KUKA KRL program: Rack_Azul_Inpicker.src, Rack_Azul_Inpicker.dat

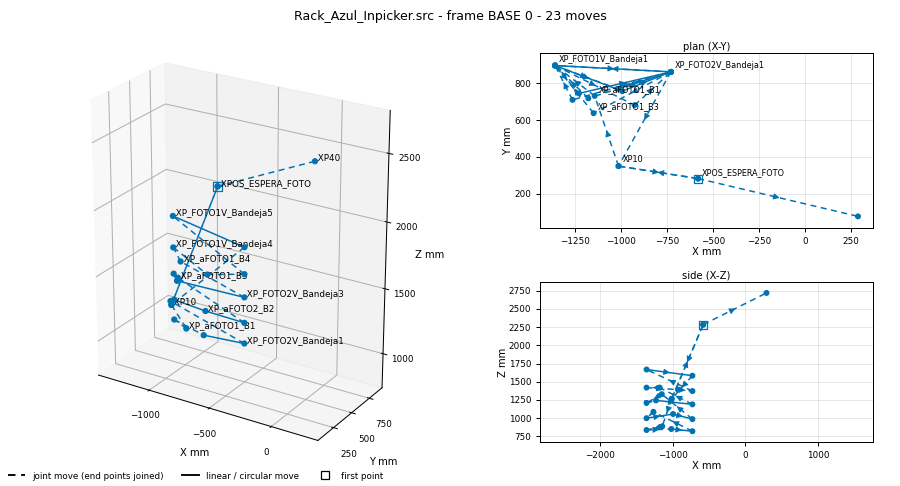
[picture p0: tool path of Rack_Azul_Inpicker.src in frame BASE 0, 23 of 23 moves have a stored position in this frame; points joined in program order, loops and branches not executed]
--- Rack_Azul_Inpicker.src ---
&ACCESS RVO1
&REL 136
&COMMENT FOTOS EN RACK AZUL
&PARAM EDITMASK = *
&PARAM TEMPLATE = C:\KRC\Roboter\Template\vorgabe
&PARAM DISKPATH = KRC:\R1\Program\MAFELEC
DEF Rack_Azul_Inpicker( )
;FOLD DECLARACION_INPICKER
DECL EKI_STATUS Ret
DECL INT InPickerStateValue
;ENDFOLD
;FOLD INI;%{PE}
  ;FOLD BASISTECH INI
    GLOBAL INTERRUPT DECL 3 WHEN $STOPMESS==TRUE DO IR_STOPM ( )
    INTERRUPT ON 3
    BAS (#INITMOV,0 )
  ;ENDFOLD (BASISTECH INI)
  ;FOLD USER INI
    ;Make your modifications here
O_LIMITS_OK=FALSE
O_LIMITS_NOK=FALSE
O_LIMIT_X=FALSE
O_LIMIT_Y=FALSE
O_LIMIT_Z=FALSE
O_LIMIT_A=FALSE
O_LIMIT_B=FALSE
O_LIMIT_C=FALSE
LIM_X=FALSE
LIM_Y=FALSE
LIM_Z=FALSE
LIM_A=FALSE
LIM_B=FALSE
LIM_C=FALSE
O_TYPE_INFO=0

  ;ENDFOLD (USER INI)
;ENDFOLD (INI)

;################################################
; PROYECTO: MAFELEC PLANTA DE BATERIAS
; ROBOT: 121_R1
; PROGRAMA: FOTO PARA CORRECCIONES EN RACK AZUL
; CREADO POR: Alejandro Company(zaisor robotics)
; FECHA: 23-NOVIEMBRE-2022
; MODIFICADO POR:
; FECHA MODIFICACION: 07-ENERO-2023
;################################################

;FOLD INICIALIZACION PUERTOS DE KRL
Ret = EKI_INIT("XML_Kuka_InPicker_1")
Ret = EKI_INIT("XML_Kuka_InPicker_2")

Ret = EKI_OPEN("XML_Kuka_InPicker_1")
Ret = EKI_OPEN("XML_Kuka_InPicker_2")

 INPICKER_Handler.DataToSend.command=0
;WAIT FOR (INPICKER_Handler.ConnectionStatus==TRUE)
;IF (INPICKER_Handler.ConnectionStatus==TRUE) THEN
;ELSE
;ENDIF

;ENDFOLD

Empujador(1,"R",FALSE)
Empujador(2,"R",FALSE)

; POSICION DE ESPERA ENTRADA RACK 2
;FOLD PTP POS_ESPERA_FOTO Vel=100 % H Tool[5]:T_Camara Base[0];%{PE}%R 8.3.48,%MKUKATPBASIS,%CMOVE,%VPTP,%P 1:PTP, 2:POS_ESPERA_FOTO, 3:, 5:100, 7:H
$BWDSTART=FALSE
PDAT_ACT=PH
FDAT_ACT=FPOS_ESPERA_FOTO
BAS(#PTP_PARAMS,100)
PTP XPOS_ESPERA_FOTO
;ENDFOLD

;ESPERA AREA 2
WAIT FOR I_ARDY_2
O_AREL_2=FALSE
RA_Bandeja_Nr=0

;FOLD PTP P10 CONT Vel=100 % M Tool[5]:T_Camara Base[0];%{PE}%R 8.3.48,%MKUKATPBASIS,%CMOVE,%VPTP,%P 1:PTP, 2:P10, 3:C_DIS, 5:100, 7:M
$BWDSTART=FALSE
PDAT_ACT=PM
FDAT_ACT=FP10
BAS(#PTP_PARAMS,100)
PTP XP10 C_DIS
;ENDFOLD
Empujador(1,"R",TRUE)
Empujador(2,"R",TRUE)

O_TYPE_RQ=TRUE
WAIT FOR (I_TYPE_INFO >= 20) AND (I_TYPE_INFO <= 26)

RA_Bandeja_Nr=I_TYPE_INFO

SWITCH RA_Bandeja_Nr

CASE 21
O_TYPE_INFO=RA_Bandeja_Nr
O_TYPE_RQ=FALSE
INICIO_FOTO1:
;FOLD PTP P_aFOTO1_B1 CONT Vel=50 % M Tool[5]:T_Camara Base[0];%{PE}%R 8.3.48,%MKUKATPBASIS,%CMOVE,%VPTP,%P 1:PTP, 2:P_aFOTO1_B1, 3:C_DIS, 5:50, 7:M
$BWDSTART=FALSE
PDAT_ACT=PM
FDAT_ACT=FP_aFOTO1_B1
BAS(#PTP_PARAMS,50)
PTP XP_aFOTO1_B1 C_DIS
;ENDFOLD
;FOLD PTP P_FOTO1V_Bandeja1 Vel=50 % M Tool[5]:T_Camara Base[0];%{PE}%R 8.3.48,%MKUKATPBASIS,%CMOVE,%VPTP,%P 1:PTP, 2:P_FOTO1V_Bandeja1, 3:, 5:50, 7:M
$BWDSTART=FALSE
PDAT_ACT=PM
FDAT_ACT=FP_FOTO1V_Bandeja1
BAS(#PTP_PARAMS,50)
PTP XP_FOTO1V_Bandeja1
;ENDFOLD
;FOLD REALIZA FOTO 1 BANDEJA 1
WAIT SEC 1.0
Fallo_nr=0
Ini1:
O_INPICKER_OK = FALSE
O_INPICKER_NOK = FALSE
SELECT_SIN=FALSE
SELECT_U1=FALSE
SELECT_U2=FALSE
SELECT_U3=FALSE
SELECT_U4=FALSE

; INICIALIZACION CAMARA PARA BANDEJA 1
 INPICKER_Handler.DataToSend.command=0
 INPICKER_Handler.DataToSend.GraspConfirmation=0
 WAIT FOR (INPICKER_Handler.DataReceived.state==0)

; Camara siempre 2
 INPICKER_Handler.DataToSend.CameraID=2

; contendor igual al numero de bandeja
 INPICKER_Handler.DataToSend.ContainerID=6
 INPICKER_Handler.DataToSend.partid=6
 INPICKER_Handler.DataToSend.GraspConfirmation=0
 WAIT SEC 0.2

; DISPARO FOTO
 INPICKER_Handler.DataToSend.command=1

; ESPERA FOTO REALIZADA
 WAIT FOR (INPICKER_Handler.DataReceived.state==15) OR (INPICKER_Handler.DataReceived.state==-1)

IF (INPICKER_Handler.DataReceived.state==-1) THEN

IF (Fallo_nr>=1) THEN
O_INPICKER_OK=FALSE
O_INPICKER_NOK=TRUE

O_TYPE_RQ = FALSE
WAIT FOR I_TYPE_INFO == 0

O_TYPE_RQ = TRUE
WAIT FOR (I_TYPE_INFO >= 1) AND (I_TYPE_INFO <= 5)

SWITCH I_TYPE_INFO

CASE 2
; #### SELECCION DESDE HMI REINTENTO FOTO ####

SELECT_NEXT=FALSE
O_INPICKER_OK=FALSE
O_INPICKER_NOK=FALSE
O_TYPE_RQ = FALSE
GOTO Ini1

CASE 3
; #### SELECCION DESDE HMI CONT SIN CORRECCION ####

SELECT_SIN=TRUE
O_INPICKER_OK=FALSE
O_INPICKER_NOK=TRUE
O_TYPE_RQ = FALSE
GOTO FIN_FOTO1

CASE 4
; #### SELECCION DESDE HMI CERRAR BANDEJA ####
; #### E IR A SIGUIENTE NIVEL             ####

SELECT_NEXT=TRUE
O_INPICKER_OK=FALSE
O_INPICKER_NOK=FALSE
O_TYPE_RQ = FALSE
GOTO FIN_FOTO1

DEFAULT
ENDSWITCH

ELSE

Fallo_nr=Fallo_nr+1
GOTO Ini1

ENDIF
ENDIF

Fin1:
 WAIT SEC 0.1
;ENDFOLD

;FOLD PTP P_aFOTO2_B1 CONT Vel=50 % M Tool[5]:T_Camara Base[0];%{PE}%R 8.3.48,%MKUKATPBASIS,%CMOVE,%VPTP,%P 1:PTP, 2:P_aFOTO2_B1, 3:C_DIS, 5:50, 7:M
$BWDSTART=FALSE
PDAT_ACT=PM
FDAT_ACT=FP_aFOTO2_B1
BAS(#PTP_PARAMS,50)
PTP XP_aFOTO2_B1 C_DIS
;ENDFOLD

;FOLD LIN P_FOTO2V_Bandeja1 Vel=0.5 m/s M Tool[5]:T_Camara Base[0];%{PE}%R 8.3.48,%MKUKATPBASIS,%CMOVE,%VLIN,%P 1:LIN, 2:P_FOTO2V_Bandeja1, 3:, 5:0.5, 7:M
$BWDSTART=FALSE
LDAT_ACT=LM
FDAT_ACT=FP_FOTO2V_Bandeja1
BAS(#CP_PARAMS,0.5)
LIN XP_FOTO2V_Bandeja1
;ENDFOLD
;FOLD REALIZA FOTO 2 BANDEJA 1 (INFERIOR)
WAIT SEC 1.0
INPICKER_Handler.DataToSend.GraspConfirmation=1

WAIT FOR (INPICKER_Handler.DataReceived.state==30) OR (INPICKER_Handler.dataReceived.state==-1)
WAIT SEC 0.5

INPICKER_Handler.DataToSend.command=0

IF (INPICKER_handler.datareceived.state==30 ) THEN

IF (INPICKER_Handler.DataReceived.ObjectsGraspable>0) THEN

O_INPICKER_OK=TRUE
O_INPICKER_NOK=FALSE

ELSE

O_INPICKER_OK=FALSE
O_INPICKER_NOK=TRUE

ENDIF

ENDIF

IF (INPICKER_handler.datareceived.state==-1 ) OR (INPICKER_Handler.DataReceived.ObjectsGraspable<=0) THEN

O_INPICKER_OK=FALSE
O_INPICKER_NOK=TRUE

O_TYPE_RQ = FALSE
WAIT FOR I_TYPE_INFO == 0

O_TYPE_RQ = TRUE
WAIT FOR (I_TYPE_INFO >= 1) AND (I_TYPE_INFO <= 5)

SWITCH I_TYPE_INFO

CASE 2
; #### SELECCION DESDE HMI REINTENTO FOTO ####

SELECT_NEXT=FALSE
O_INPICKER_OK=FALSE
O_INPICKER_NOK=FALSE
O_TYPE_RQ = FALSE

IF (INPICKER_Handler.DataReceived.ObjectsGraspable>0)THEN
ELSE
GOTO INICIO_FOTO1
ENDIF

WAIT FOR (INPICKER_Handler.DataReceived.state==0)
GOTO INICIO_FOTO1

CASE 3
; #### SELECCION DESDE HMI CONT SIN CORRECCION ####

SELECT_NEXT=FALSE
O_TYPE_RQ = FALSE

CASE 4
; #### SELECCION DESDE HMI CERRAR BANDEJA ####
; #### E IR A SIGUIENTE NIVEL             ####

SELECT_NEXT=TRUE
O_INPICKER_OK=FALSE
O_INPICKER_NOK=FALSE
O_TYPE_RQ = FALSE

DEFAULT
ENDSWITCH

ENDIF

;ENDFOLD
;FOLD ACTUALIZA BASE DE DESCARGA
FRAMEAUX={X 0,Y 0,Z 0,A 0,B 0,C 0}
FRAME_POS={X 0,Y 0,Z 0,A 0,B 0,C 0}

FRAMEAUX=INPICKER_Handler.DataReceived.PartsToGrasp0.Position
FRAME_POS.x=(FRAMEAUX.x/10)
FRAME_POS.y=(FRAMEAUX.y/10)
FRAME_POS.z=(FRAMEAUX.z/10)
FRAME_POS.a=(FRAMEAUX.a/10)
FRAME_POS.b=(FRAMEAUX.b/10)
FRAME_POS.c=(FRAMEAUX.c/10)

IF FRAME_POS.A < 180.0 THEN
FRAME_POS.A = FRAME_POS.A + 360
ENDIF
IF FRAME_POS.B < 180.0 THEN
FRAME_POS.B = FRAME_POS.B + 360
ENDIF
IF FRAME_POS.A > 180.0 THEN
FRAME_POS.A = FRAME_POS.A - 360
ENDIF
IF FRAME_POS.B > 180.0 THEN
FRAME_POS.B = FRAME_POS.B - 360
ENDIF

FRAME_POS.C = FRAME_POS.C - 360

;ENDFOLD
;FOLD CONTROL LIMITES DE VISION
CTRL_limites()
;ENDFOLD
;FOLD DECISION RESULTADOS EVALUACION BANDEJA 1

IF (O_INPICKER_OK==FALSE) AND (O_INPICKER_NOK==TRUE) THEN
SELECT_NEXT=FALSE
O_TYPE_RQ = FALSE
GOTO FIN_FOTO1
ENDIF


IF (O_LIMITS_OK==FALSE) AND (O_LIMITS_NOK==TRUE) THEN

O_TYPE_RQ = FALSE
WAIT FOR I_TYPE_INFO == 0

O_TYPE_RQ = TRUE
WAIT FOR (I_TYPE_INFO >= 1) AND (I_TYPE_INFO <= 5)

SWITCH I_TYPE_INFO

CASE 2
; #### SELECCION DESDE HMI REINTENTO FOTO ####

SELECT_NEXT=FALSE
O_TYPE_RQ = FALSE
O_LIMITS_OK = FALSE
O_LIMITS_NOK = FALSE
O_LIMIT_X = FALSE
O_LIMIT_Y = FALSE
O_LIMIT_Z = FALSE
O_LIMIT_A = FALSE
O_LIMIT_B = FALSE
O_LIMIT_C = FALSE

GOTO INICIO_FOTO1

CASE 3
; #### SELECCION DESDE HMI CONT SIN CORRECCION ####

SELECT_NEXT=FALSE
O_TYPE_RQ = FALSE

CASE 4
; #### SELECCION DESDE HMI CERRAR BANDEJA ####
; #### E IR A SIGUIENTE NIVEL             ####

SELECT_NEXT=TRUE
O_TYPE_RQ = FALSE
O_LIMITS_OK = FALSE
O_LIMITS_NOK = FALSE
O_LIMIT_X = FALSE
O_LIMIT_Y = FALSE
O_LIMIT_Z = FALSE
O_LIMIT_A = FALSE
O_LIMIT_B = FALSE
O_LIMIT_C = FALSE

DEFAULT

HALT
HALT
HALT
ENDSWITCH

ENDIF

NO_TYPE_LBL:
;ENDFOLD
FIN_FOTO1:

CASE 22
O_TYPE_INFO=RA_Bandeja_Nr
O_TYPE_RQ=FALSE
INICIO_FOTO2:
;FOLD PTP P_aFOTO1_B2 Vel=50 % M Tool[5]:T_Camara Base[0];%{PE}%R 8.3.48,%MKUKATPBASIS,%CMOVE,%VPTP,%P 1:PTP, 2:P_aFOTO1_B2, 3:, 5:50, 7:M
$BWDSTART=FALSE
PDAT_ACT=PM
FDAT_ACT=FP_aFOTO1_B2
BAS(#PTP_PARAMS,50)
PTP XP_aFOTO1_B2
;ENDFOLD
;FOLD PTP P_FOTO1V_Bandeja2 Vel=50 % M Tool[5]:T_Camara Base[0];%{PE}%R 8.3.48,%MKUKATPBASIS,%CMOVE,%VPTP,%P 1:PTP, 2:P_FOTO1V_Bandeja2, 3:, 5:50, 7:M
$BWDSTART=FALSE
PDAT_ACT=PM
FDAT_ACT=FP_FOTO1V_Bandeja2
BAS(#PTP_PARAMS,50)
PTP XP_FOTO1V_Bandeja2
;ENDFOLD
;FOLD REALIZA FOTO 1 BANDEJA 2
WAIT SEC 1.0
Fallo_nr=0
Ini2:
O_INPICKER_OK = FALSE
O_INPICKER_NOK = FALSE
SELECT_SIN=FALSE
SELECT_U1=FALSE
SELECT_U2=FALSE
SELECT_U3=FALSE
SELECT_U4=FALSE

; INICIALIZACION CAMARA PARA BANDEJA 2
 INPICKER_Handler.DataToSend.command=0
 INPICKER_Handler.DataToSend.GraspConfirmation=0
 WAIT FOR (INPICKER_Handler.DataReceived.state==0)

; Camara siempre 2
 INPICKER_Handler.DataToSend.CameraID=2

; contendor igual al numero de bandeja
 INPICKER_Handler.DataToSend.ContainerID=7
 INPICKER_Handler.DataToSend.partid=7
 INPICKER_Handler.DataToSend.GraspConfirmation=0
 WAIT SEC 0.2

; DISPARO FOTO
 INPICKER_Handler.DataToSend.command=1

; ESPERA FOTO REALIZADA
 WAIT FOR (INPICKER_Handler.DataReceived.state==15) OR (INPICKER_Handler.DataReceived.state==-1)

IF (INPICKER_Handler.DataReceived.state==-1) THEN

IF (Fallo_nr>=1) THEN
O_INPICKER_OK=FALSE
O_INPICKER_NOK=TRUE

O_TYPE_RQ = FALSE
WAIT FOR I_TYPE_INFO == 0

O_TYPE_RQ = TRUE
WAIT FOR (I_TYPE_INFO >= 1) AND (I_TYPE_INFO <= 5)

SWITCH I_TYPE_INFO

CASE 2
; #### SELECCION DESDE HMI REINTENTO FOTO ####

SELECT_NEXT=FALSE
O_INPICKER_OK=FALSE
O_INPICKER_NOK=FALSE
O_TYPE_RQ = FALSE
GOTO Ini2

CASE 3
; #### SELECCION DESDE HMI CONT SIN CORRECCION ####

SELECT_SIN=TRUE
O_INPICKER_OK=FALSE
O_INPICKER_NOK=TRUE
O_TYPE_RQ = FALSE
GOTO FIN_FOTO2

CASE 4
; #### SELECCION DESDE HMI CERRAR BANDEJA ####
; #### E IR A SIGUIENTE NIVEL             ####

SELECT_NEXT=TRUE
O_INPICKER_OK=FALSE
O_INPICKER_NOK=FALSE
O_TYPE_RQ = FALSE
GOTO FIN_FOTO2

DEFAULT
ENDSWITCH

ELSE

Fallo_nr=Fallo_nr+1
GOTO Ini2

ENDIF
ENDIF

Fin2:
 WAIT SEC 0.1
;ENDFOLD

;FOLD LIN P_aFOTO2_B2 Vel=0.3 m/s M Tool[5]:T_Camara Base[0];%{PE}%R 8.3.48,%MKUKATPBASIS,%CMOVE,%VLIN,%P 1:LIN, 2:P_aFOTO2_B2, 3:, 5:0.3, 7:M
$BWDSTART=FALSE
LDAT_ACT=LM
FDAT_ACT=FP_aFOTO2_B2
BAS(#CP_PARAMS,0.3)
LIN XP_aFOTO2_B2
;ENDFOLD

;FOLD LIN P_FOTO2V_Bandeja2 Vel=0.5 m/s M Tool[5]:T_Camara Base[0];%{PE}%R 8.3.48,%MKUKATPBASIS,%CMOVE,%VLIN,%P 1:LIN, 2:P_FOTO2V_Bandeja2, 3:, 5:0.5, 7:M
$BWDSTART=FALSE
LDAT_ACT=LM
FDAT_ACT=FP_FOTO2V_Bandeja2
BAS(#CP_PARAMS,0.5)
LIN XP_FOTO2V_Bandeja2
;ENDFOLD
;FOLD REALIZA FOTO 2 BANDEJA 2
WAIT SEC 1.0
INPICKER_Handler.DataToSend.GraspConfirmation=1

WAIT FOR (INPICKER_Handler.DataReceived.state==30) OR (INPICKER_Handler.dataReceived.state==-1)

WAIT SEC 0.5

INPICKER_Handler.DataToSend.command=0

IF (INPICKER_handler.datareceived.state==30 ) THEN

IF (INPICKER_Handler.DataReceived.ObjectsGraspable>0) THEN

O_INPICKER_OK=TRUE
O_INPICKER_NOK=FALSE

ELSE

O_INPICKER_OK=FALSE
O_INPICKER_NOK=TRUE

ENDIF

ENDIF

IF (INPICKER_handler.datareceived.state==-1 ) OR (INPICKER_Handler.DataReceived.ObjectsGraspable<=0) THEN

O_INPICKER_OK=FALSE
O_INPICKER_NOK=TRUE

O_TYPE_RQ = FALSE
WAIT FOR I_TYPE_INFO == 0

O_TYPE_RQ = TRUE
WAIT FOR (I_TYPE_INFO >= 1) AND (I_TYPE_INFO <= 5)

SWITCH I_TYPE_INFO

CASE 2
; #### SELECCION DESDE HMI REINTENTO FOTO ####

SELECT_NEXT=FALSE
O_INPICKER_OK=FALSE
O_INPICKER_NOK=FALSE
O_TYPE_RQ = FALSE

IF (INPICKER_Handler.DataReceived.ObjectsGraspable>0)THEN
ELSE
GOTO INICIO_FOTO2
ENDIF

WAIT FOR (INPICKER_Handler.DataReceived.state==0)
GOTO INICIO_FOTO2

CASE 3
; #### SELECCION DESDE HMI CONT SIN CORRECCION ####

SELECT_NEXT=FALSE
O_TYPE_RQ = FALSE

CASE 4
; #### SELECCION DESDE HMI CERRAR BANDEJA ####
; #### E IR A SIGUIENTE NIVEL             ####

SELECT_NEXT=TRUE
O_INPICKER_OK=FALSE
O_INPICKER_NOK=FALSE
O_TYPE_RQ = FALSE

DEFAULT
ENDSWITCH

ENDIF

;ENDFOLD
;FOLD ACTUALIZA BASE DE DESCARGA
FRAMEAUX={X 0,Y 0,Z 0,A 0,B 0,C 0}
FRAME_POS={X 0,Y 0,Z 0,A 0,B 0,C 0}

FRAMEAUX=INPICKER_Handler.DataReceived.PartsToGrasp0.Position
FRAME_POS.x=(FRAMEAUX.x/10)
FRAME_POS.y=(FRAMEAUX.y/10)
FRAME_POS.z=(FRAMEAUX.z/10)
FRAME_POS.a=(FRAMEAUX.a/10)
FRAME_POS.b=(FRAMEAUX.b/10)
FRAME_POS.c=(FRAMEAUX.c/10)

IF FRAME_POS.A < 180.0 THEN
FRAME_POS.A = FRAME_POS.A + 360
ENDIF
IF FRAME_POS.B < 180.0 THEN
FRAME_POS.B = FRAME_POS.B + 360
ENDIF
IF FRAME_POS.A > 180.0 THEN
FRAME_POS.A = FRAME_POS.A - 360
ENDIF
IF FRAME_POS.B > 180.0 THEN
FRAME_POS.B = FRAME_POS.B - 360
ENDIF
FRAME_POS.C = FRAME_POS.C - 360
;ENDFOLD
;FOLD CONTROL LIMITES DE VISION
CTRL_limites()
;ENDFOLD
;FOLD DECISION RESULTADOS EVALUACION BANDEJA 2

IF (O_INPICKER_OK==FALSE) AND (O_INPICKER_NOK==TRUE) THEN
SELECT_NEXT=FALSE
O_TYPE_RQ = FALSE
GOTO FIN_FOTO2
ENDIF



IF (O_LIMITS_OK==FALSE) AND (O_LIMITS_NOK==TRUE) THEN

O_TYPE_RQ = FALSE
WAIT FOR I_TYPE_INFO == 0

O_TYPE_RQ = TRUE
WAIT FOR (I_TYPE_INFO >= 1) AND (I_TYPE_INFO <= 5)

SWITCH I_TYPE_INFO

CASE 2
; #### SELECCION DESDE HMI REINTENTO FOTO ####

SELECT_NEXT=FALSE
O_TYPE_RQ = FALSE
O_LIMITS_OK = FALSE
O_LIMITS_NOK = FALSE
O_LIMIT_X = FALSE
O_LIMIT_Y = FALSE
O_LIMIT_Z = FALSE
O_LIMIT_A = FALSE
O_LIMIT_B = FALSE
O_LIMIT_C = FALSE

GOTO INICIO_FOTO2

CASE 3
; #### SELECCION DESDE HMI CONT SIN CORRECCION ####

SELECT_NEXT=FALSE
O_TYPE_RQ = FALSE

CASE 4
; #### SELECCION DESDE HMI CERRAR BANDEJA ####
; #### E IR A SIGUIENTE NIVEL             ####

SELECT_NEXT=TRUE
O_TYPE_RQ = FALSE
O_LIMITS_OK = FALSE
O_LIMITS_NOK = FALSE
O_LIMIT_X = FALSE
O_LIMIT_Y = FALSE
O_LIMIT_Z = FALSE
O_LIMIT_A = FALSE
O_LIMIT_B = FALSE
O_LIMIT_C = FALSE

DEFAULT

HALT
HALT
HALT
ENDSWITCH

ENDIF

;ENDFOLD
FIN_FOTO2:

CASE 23
O_TYPE_RQ=FALSE
O_TYPE_INFO=RA_Bandeja_Nr
INICIO_FOTO3:
;FOLD PTP P_aFOTO1_B3 CONT Vel=50 % M Tool[5]:T_Camara Base[0];%{PE}%R 8.3.48,%MKUKATPBASIS,%CMOVE,%VPTP,%P 1:PTP, 2:P_aFOTO1_B3, 3:C_DIS, 5:50, 7:M
$BWDSTART=FALSE
PDAT_ACT=PM
FDAT_ACT=FP_aFOTO1_B3
BAS(#PTP_PARAMS,50)
PTP XP_aFOTO1_B3 C_DIS
;ENDFOLD
;FOLD PTP P_FOTO1V_Bandeja3 Vel=50 % M Tool[5]:T_Camara Base[0];%{PE}%R 8.3.48,%MKUKATPBASIS,%CMOVE,%VPTP,%P 1:PTP, 2:P_FOTO1V_Bandeja3, 3:, 5:50, 7:M
$BWDSTART=FALSE
PDAT_ACT=PM
FDAT_ACT=FP_FOTO1V_Bandeja3
BAS(#PTP_PARAMS,50)
PTP XP_FOTO1V_Bandeja3
;ENDFOLD
;FOLD REALIZA FOTO 1 BANDEJA 3
WAIT SEC 1.0
Fallo_nr=0
Ini3:
O_INPICKER_OK = FALSE
O_INPICKER_NOK = FALSE
SELECT_SIN=FALSE
SELECT_U1=FALSE
SELECT_U2=FALSE
SELECT_U3=FALSE
SELECT_U4=FALSE

; INICIALIZACION CAMARA PARA BANDEJA 3
 INPICKER_Handler.DataToSend.command=0
 INPICKER_Handler.DataToSend.GraspConfirmation=0
 WAIT FOR (INPICKER_Handler.DataReceived.state==0)

; Camara siempre 2
 INPICKER_Handler.DataToSend.CameraID=2

; contendor igual al numero de bandeja
 INPICKER_Handler.DataToSend.ContainerID=8
 INPICKER_Handler.DataToSend.partid=8
 INPICKER_Handler.DataToSend.GraspConfirmation=0
 WAIT SEC 0.2

; DISPARO FOTO
 INPICKER_Handler.DataToSend.command=1

; ESPERA FOTO REALIZADA
 WAIT FOR (INPICKER_Handler.DataReceived.state==15) OR (INPICKER_Handler.DataReceived.state==-1)

IF (INPICKER_Handler.DataReceived.state==-1) THEN

IF (Fallo_nr>=1) THEN
O_INPICKER_OK=FALSE
O_INPICKER_NOK=TRUE

O_TYPE_RQ = FALSE
WAIT FOR I_TYPE_INFO == 0

O_TYPE_RQ = TRUE
WAIT FOR (I_TYPE_INFO >= 1) AND (I_TYPE_INFO <= 5)

SWITCH I_TYPE_INFO

CASE 2
; #### SELECCION DESDE HMI REINTENTO FOTO ####

SELECT_NEXT=FALSE
O_INPICKER_OK=FALSE
O_INPICKER_NOK=FALSE
O_TYPE_RQ = FALSE
GOTO Ini3

CASE 3
; #### SELECCION DESDE HMI CONT SIN CORRECCION ####

SELECT_SIN=TRUE
O_INPICKER_OK=FALSE
O_INPICKER_NOK=TRUE
O_TYPE_RQ = FALSE
GOTO FIN_FOTO3

CASE 4
; #### SELECCION DESDE HMI CERRAR BANDEJA ####
; #### E IR A SIGUIENTE NIVEL             ####

SELECT_NEXT=TRUE
O_INPICKER_OK=FALSE
O_INPICKER_NOK=FALSE
O_TYPE_RQ = FALSE
GOTO FIN_FOTO3

DEFAULT
ENDSWITCH

ELSE

Fallo_nr=Fallo_nr+1
GOTO Ini3

ENDIF
ENDIF

Fin3:
 WAIT SEC 0.1
;ENDFOLD

;FOLD PTP P_aFOTO2_B3 CONT Vel=50 % M Tool[5]:T_Camara Base[0];%{PE}%R 8.3.48,%MKUKATPBASIS,%CMOVE,%VPTP,%P 1:PTP, 2:P_aFOTO2_B3, 3:C_DIS, 5:50, 7:M
$BWDSTART=FALSE
PDAT_ACT=PM
FDAT_ACT=FP_aFOTO2_B3
BAS(#PTP_PARAMS,50)
PTP XP_aFOTO2_B3 C_DIS
;ENDFOLD

;FOLD LIN P_FOTO2V_Bandeja3 Vel=0.3 m/s M Tool[5]:T_Camara Base[0];%{PE}%R 8.3.48,%MKUKATPBASIS,%CMOVE,%VLIN,%P 1:LIN, 2:P_FOTO2V_Bandeja3, 3:, 5:0.3, 7:M
$BWDSTART=FALSE
LDAT_ACT=LM
FDAT_ACT=FP_FOTO2V_Bandeja3
BAS(#CP_PARAMS,0.3)
LIN XP_FOTO2V_Bandeja3
;ENDFOLD
;FOLD REALIZA FOTO 2 BANDEJA 3
WAIT SEC 1.0
INPICKER_Handler.DataToSend.GraspConfirmation=1

WAIT FOR (INPICKER_Handler.DataReceived.state==30) OR (INPICKER_Handler.dataReceived.state==-1)

WAIT SEC 0.5

INPICKER_Handler.DataToSend.command=0

IF (INPICKER_handler.datareceived.state==30 ) THEN

IF (INPICKER_Handler.DataReceived.ObjectsGraspable>0) THEN

O_INPICKER_OK=TRUE
O_INPICKER_NOK=FALSE

ELSE

O_INPICKER_OK=FALSE
O_INPICKER_NOK=TRUE

ENDIF

ENDIF

IF (INPICKER_handler.datareceived.state==-1 ) OR (INPICKER_Handler.DataReceived.ObjectsGraspable<=0) THEN

O_INPICKER_OK=FALSE
O_INPICKER_NOK=TRUE

O_TYPE_RQ = FALSE
WAIT FOR I_TYPE_INFO == 0

O_TYPE_RQ = TRUE
WAIT FOR (I_TYPE_INFO >= 1) AND (I_TYPE_INFO <= 5)

SWITCH I_TYPE_INFO

CASE 2
; #### SELECCION DESDE HMI REINTENTO FOTO ####

SELECT_NEXT=FALSE
O_INPICKER_OK=FALSE
O_INPICKER_NOK=FALSE
O_TYPE_RQ = FALSE

IF (INPICKER_Handler.DataReceived.ObjectsGraspable>0)THEN
ELSE
GOTO INICIO_FOTO3
ENDIF

WAIT FOR (INPICKER_Handler.DataReceived.state==0)
GOTO INICIO_FOTO3

CASE 3
; #### SELECCION DESDE HMI CONT SIN CORRECCION ####

SELECT_NEXT=FALSE
O_TYPE_RQ = FALSE

CASE 4
; #### SELECCION DESDE HMI CERRAR BANDEJA ####
; #### E IR A SIGUIENTE NIVEL             ####

SELECT_NEXT=TRUE
O_INPICKER_OK=FALSE
O_INPICKER_NOK=FALSE
O_TYPE_RQ = FALSE

DEFAULT
ENDSWITCH

ENDIF

;ENDFOLD
;FOLD ACTUALIZA BASE DE DESCARGA
FRAMEAUX={X 0,Y 0,Z 0,A 0,B 0,C 0}
FRAME_POS={X 0,Y 0,Z 0,A 0,B 0,C 0}

FRAMEAUX=INPICKER_Handler.DataReceived.PartsToGrasp0.Position
FRAME_POS.x=(FRAMEAUX.x/10)
FRAME_POS.y=(FRAMEAUX.y/10)
FRAME_POS.z=(FRAMEAUX.z/10)
FRAME_POS.a=(FRAMEAUX.a/10)
FRAME_POS.b=(FRAMEAUX.b/10)
FRAME_POS.c=(FRAMEAUX.c/10)

IF FRAME_POS.A < 180.0 THEN
FRAME_POS.A = FRAME_POS.A + 360
ENDIF
IF FRAME_POS.B < 180.0 THEN
FRAME_POS.B = FRAME_POS.B + 360
ENDIF
IF FRAME_POS.A > 180.0 THEN
FRAME_POS.A = FRAME_POS.A - 360
ENDIF
IF FRAME_POS.B > 180.0 THEN
FRAME_POS.B = FRAME_POS.B - 360
ENDIF
FRAME_POS.C = FRAME_POS.C - 360
;ENDFOLD
;FOLD CONTROL LIMITES DE VISION
CTRL_limites()
;ENDFOLD
;FOLD DECISION RESULTADOS EVALUACION BANDEJA 3

IF (O_INPICKER_OK==FALSE) AND (O_INPICKER_NOK==TRUE) THEN
SELECT_NEXT=FALSE
O_TYPE_RQ = FALSE
GOTO FIN_FOTO3
ENDIF


IF (O_LIMITS_OK==FALSE) AND (O_LIMITS_NOK==TRUE) THEN

O_TYPE_RQ = FALSE
WAIT FOR I_TYPE_INFO == 0

O_TYPE_RQ = TRUE
WAIT FOR (I_TYPE_INFO >= 1) AND (I_TYPE_INFO <= 5)

SWITCH I_TYPE_INFO

CASE 2
; #### SELECCION DESDE HMI REINTENTO FOTO ####

SELECT_NEXT=FALSE
O_TYPE_RQ = FALSE
O_LIMITS_OK = FALSE
O_LIMITS_NOK = FALSE
O_LIMIT_X = FALSE
O_LIMIT_Y = FALSE
O_LIMIT_Z = FALSE
O_LIMIT_A = FALSE
O_LIMIT_B = FALSE
O_LIMIT_C = FALSE

GOTO INICIO_FOTO3

CASE 3
; #### SELECCION DESDE HMI CONT SIN CORRECCION ####

SELECT_NEXT=FALSE
O_TYPE_RQ = FALSE

CASE 4
; #### SELECCION DESDE HMI CERRAR BANDEJA ####
; #### E IR A SIGUIENTE NIVEL             ####

SELECT_NEXT=TRUE
O_TYPE_RQ = FALSE
O_LIMITS_OK = FALSE
O_LIMITS_NOK = FALSE
O_LIMIT_X = FALSE
O_LIMIT_Y = FALSE
O_LIMIT_Z = FALSE
O_LIMIT_A = FALSE
O_LIMIT_B = FALSE
O_LIMIT_C = FALSE

DEFAULT

HALT
HALT
HALT
ENDSWITCH

ENDIF
;ENDFOLD
FIN_FOTO3:

CASE 24
O_TYPE_RQ=FALSE
O_TYPE_INFO=RA_Bandeja_Nr
INICIO_FOTO4:
;FOLD PTP P_aFOTO1_B4 CONT Vel=50 % M Tool[5]:T_Camara Base[0];%{PE}%R 8.3.48,%MKUKATPBASIS,%CMOVE,%VPTP,%P 1:PTP, 2:P_aFOTO1_B4, 3:C_DIS, 5:50, 7:M
$BWDSTART=FALSE
PDAT_ACT=PM
FDAT_ACT=FP_aFOTO1_B4
BAS(#PTP_PARAMS,50)
PTP XP_aFOTO1_B4 C_DIS
;ENDFOLD
;FOLD PTP P_FOTO1V_Bandeja4 Vel=50 % M Tool[5]:T_Camara Base[0];%{PE}%R 8.3.48,%MKUKATPBASIS,%CMOVE,%VPTP,%P 1:PTP, 2:P_FOTO1V_Bandeja4, 3:, 5:50, 7:M
$BWDSTART=FALSE
PDAT_ACT=PM
FDAT_ACT=FP_FOTO1V_Bandeja4
BAS(#PTP_PARAMS,50)
PTP XP_FOTO1V_Bandeja4
;ENDFOLD
;FOLD REALIZA FOTO 1 BANDEJA 4
WAIT SEC 1.0
Fallo_nr=0
Ini4:
O_INPICKER_OK = FALSE
O_INPICKER_NOK = FALSE
SELECT_SIN=FALSE
SELECT_U1=FALSE
SELECT_U2=FALSE
SELECT_U3=FALSE
SELECT_U4=FALSE

; INICIALIZACION CAMARA PARA BANDEJA 1
 INPICKER_Handler.DataToSend.command=0
 INPICKER_Handler.DataToSend.GraspConfirmation=0
 WAIT FOR (INPICKER_Handler.DataReceived.state==0)

; Camara siempre 2
 INPICKER_Handler.DataToSend.CameraID=2

; contendor igual al numero de bandeja
 INPICKER_Handler.DataToSend.ContainerID=9
 INPICKER_Handler.DataToSend.partid=9
 INPICKER_Handler.DataToSend.GraspConfirmation=0
 WAIT SEC 0.2

; DISPARO FOTO
 INPICKER_Handler.DataToSend.command=1

; ESPERA FOTO REALIZADA
 WAIT FOR (INPICKER_Handler.DataReceived.state==15) OR (INPICKER_Handler.DataReceived.state==-1)

IF (INPICKER_Handler.DataReceived.state==-1) THEN

IF (Fallo_nr>=1) THEN
O_INPICKER_OK=FALSE
O_INPICKER_NOK=TRUE

O_TYPE_RQ = FALSE
WAIT FOR I_TYPE_INFO == 0

O_TYPE_RQ = TRUE
WAIT FOR (I_TYPE_INFO >= 1) AND (I_TYPE_INFO <= 5)

SWITCH I_TYPE_INFO

CASE 2
; #### SELECCION DESDE HMI REINTENTO FOTO ####

SELECT_NEXT=FALSE
O_INPICKER_OK=FALSE
O_INPICKER_NOK=FALSE
O_TYPE_RQ = FALSE
GOTO Ini4

CASE 3
; #### SELECCION DESDE HMI CONT SIN CORRECCION ####

SELECT_SIN=TRUE
O_INPICKER_OK=FALSE
O_INPICKER_NOK=TRUE
O_TYPE_RQ = FALSE
GOTO FIN_FOTO4

CASE 4
; #### SELECCION DESDE HMI CERRAR BANDEJA ####
; #### E IR A SIGUIENTE NIVEL             ####

SELECT_NEXT=TRUE
O_INPICKER_OK=FALSE
O_INPICKER_NOK=FALSE
O_TYPE_RQ = FALSE
GOTO FIN_FOTO4

DEFAULT
ENDSWITCH

ELSE

Fallo_nr=Fallo_nr+1
GOTO Ini4

ENDIF
ENDIF

Fin4:
 WAIT SEC 0.1
;ENDFOLD

;FOLD PTP P_aFOTO2_B4 CONT Vel=50 % M Tool[5]:T_Camara Base[0];%{PE}%R 8.3.48,%MKUKATPBASIS,%CMOVE,%VPTP,%P 1:PTP, 2:P_aFOTO2_B4, 3:C_DIS, 5:50, 7:M
$BWDSTART=FALSE
PDAT_ACT=PM
FDAT_ACT=FP_aFOTO2_B4
BAS(#PTP_PARAMS,50)
PTP XP_aFOTO2_B4 C_DIS
;ENDFOLD

;FOLD PTP P_FOTO2V_Bandeja4 Vel=50 % M Tool[5]:T_Camara Base[0];%{PE}%R 8.3.48,%MKUKATPBASIS,%CMOVE,%VPTP,%P 1:PTP, 2:P_FOTO2V_Bandeja4, 3:, 5:50, 7:M
$BWDSTART=FALSE
PDAT_ACT=PM
FDAT_ACT=FP_FOTO2V_Bandeja4
BAS(#PTP_PARAMS,50)
PTP XP_FOTO2V_Bandeja4
;ENDFOLD
;FOLD REALIZA FOTO 2 BANDEJA 4
WAIT SEC 1.0
INPICKER_Handler.DataToSend.GraspConfirmation=1

WAIT FOR (INPICKER_Handler.DataReceived.state==30) OR (INPICKER_Handler.dataReceived.state==-1)

WAIT SEC 0.5

INPICKER_Handler.DataToSend.command=0

IF (INPICKER_handler.datareceived.state==30 ) THEN

IF (INPICKER_Handler.DataReceived.ObjectsGraspable>0) THEN

O_INPICKER_OK=TRUE
O_INPICKER_NOK=FALSE

ELSE

O_INPICKER_OK=FALSE
O_INPICKER_NOK=TRUE

ENDIF

ENDIF

IF (INPICKER_handler.datareceived.state==-1 ) OR (INPICKER_Handler.DataReceived.ObjectsGraspable<=0) THEN

O_INPICKER_OK=FALSE
O_INPICKER_NOK=TRUE

O_TYPE_RQ = FALSE
WAIT FOR I_TYPE_INFO == 0

O_TYPE_RQ = TRUE
WAIT FOR (I_TYPE_INFO >= 1) AND (I_TYPE_INFO <= 5)

SWITCH I_TYPE_INFO

CASE 2
; #### SELECCION DESDE HMI REINTENTO FOTO ####

SELECT_NEXT=FALSE
O_INPICKER_OK=FALSE
O_INPICKER_NOK=FALSE
O_TYPE_RQ = FALSE

IF (INPICKER_Handler.DataReceived.ObjectsGraspable>0)THEN
ELSE
GOTO INICIO_FOTO4
ENDIF

WAIT FOR (INPICKER_Handler.DataReceived.state==0)
GOTO INICIO_FOTO4

CASE 3
; #### SELECCION DESDE HMI CONT SIN CORRECCION ####

SELECT_NEXT=FALSE
O_TYPE_RQ = FALSE

CASE 4
; #### SELECCION DESDE HMI CERRAR BANDEJA ####
; #### E IR A SIGUIENTE NIVEL             ####

SELECT_NEXT=TRUE
O_INPICKER_OK=FALSE
O_INPICKER_NOK=FALSE
O_TYPE_RQ = FALSE

DEFAULT
ENDSWITCH

ENDIF

;ENDFOLD
;FOLD ACTUALIZA BASE DE DESCARGA
FRAMEAUX={X 0,Y 0,Z 0,A 0,B 0,C 0}
FRAME_POS={X 0,Y 0,Z 0,A 0,B 0,C 0}

FRAMEAUX=INPICKER_Handler.DataReceived.PartsToGrasp0.Position
FRAME_POS.x=(FRAMEAUX.x/10)
FRAME_POS.y=(FRAMEAUX.y/10)
FRAME_POS.z=(FRAMEAUX.z/10)
FRAME_POS.a=(FRAMEAUX.a/10)
FRAME_POS.b=(FRAMEAUX.b/10)
FRAME_POS.c=(FRAMEAUX.c/10)

IF FRAME_POS.A < 180.0 THEN
FRAME_POS.A = FRAME_POS.A + 360
ENDIF
IF FRAME_POS.B < 180.0 THEN
FRAME_POS.B = FRAME_POS.B + 360
ENDIF
IF FRAME_POS.A > 180.0 THEN
FRAME_POS.A = FRAME_POS.A - 360
ENDIF
IF FRAME_POS.B > 180.0 THEN
FRAME_POS.B = FRAME_POS.B - 360
ENDIF
FRAME_POS.C = FRAME_POS.C - 360
;ENDFOLD
;FOLD CONTROL LIMITES DE VISION
CTRL_limites()
;ENDFOLD
;FOLD DECISION RESULTADOS EVALUACION BANDEJA 4

IF (O_INPICKER_OK==FALSE) AND (O_INPICKER_NOK==TRUE) THEN
SELECT_NEXT=FALSE
O_TYPE_RQ = FALSE
GOTO FIN_FOTO4
ENDIF


IF (O_LIMITS_OK==FALSE) AND (O_LIMITS_NOK==TRUE) THEN

O_TYPE_RQ = FALSE
WAIT FOR I_TYPE_INFO == 0

O_TYPE_RQ = TRUE
WAIT FOR (I_TYPE_INFO >= 1) AND (I_TYPE_INFO <= 5)

SWITCH I_TYPE_INFO

CASE 2
; #### SELECCION DESDE HMI REINTENTO FOTO ####

SELECT_NEXT=FALSE
O_TYPE_RQ = FALSE
O_LIMITS_OK = FALSE
O_LIMITS_NOK = FALSE
O_LIMIT_X = FALSE
O_LIMIT_Y = FALSE
O_LIMIT_Z = FALSE
O_LIMIT_A = FALSE
O_LIMIT_B = FALSE
O_LIMIT_C = FALSE

GOTO INICIO_FOTO4

CASE 3
; #### SELECCION DESDE HMI CONT SIN CORRECCION ####

SELECT_NEXT=FALSE
O_TYPE_RQ = FALSE

CASE 4
; #### SELECCION DESDE HMI CERRAR BANDEJA ####
; #### E IR A SIGUIENTE NIVEL             ####

SELECT_NEXT=TRUE
O_TYPE_RQ = FALSE
O_LIMITS_OK = FALSE
O_LIMITS_NOK = FALSE
O_LIMIT_X = FALSE
O_LIMIT_Y = FALSE
O_LIMIT_Z = FALSE
O_LIMIT_A = FALSE
O_LIMIT_B = FALSE
O_LIMIT_C = FALSE

DEFAULT

HALT
HALT
HALT
ENDSWITCH

ENDIF
;ENDFOLD
FIN_FOTO4:

CASE 25
O_TYPE_RQ=FALSE
O_TYPE_INFO=RA_Bandeja_Nr
INICIO_FOTO5:
;FOLD PTP P_FOTO1V_Bandeja5 Vel=50 % M Tool[5]:T_Camara Base[0];%{PE}%R 8.3.48,%MKUKATPBASIS,%CMOVE,%VPTP,%P 1:PTP, 2:P_FOTO1V_Bandeja5, 3:, 5:50, 7:M
$BWDSTART=FALSE
PDAT_ACT=PM
FDAT_ACT=FP_FOTO1V_Bandeja5
BAS(#PTP_PARAMS,50)
PTP XP_FOTO1V_Bandeja5
;ENDFOLD
;FOLD REALIZA FOTO 1 BANDEJA 5
WAIT SEC 1.0
Fallo_nr=0
Ini5:
O_INPICKER_OK = FALSE
O_INPICKER_NOK = FALSE
SELECT_SIN=FALSE
SELECT_U1=FALSE
SELECT_U2=FALSE
SELECT_U3=FALSE
SELECT_U4=FALSE

; INICIALIZACION CAMARA PARA BANDEJA 5
 INPICKER_Handler.DataToSend.command=0
 INPICKER_Handler.DataToSend.GraspConfirmation=0
 WAIT FOR (INPICKER_Handler.DataReceived.state==0)

; Camara siempre 2
 INPICKER_Handler.DataToSend.CameraID=2

; contendor igual al numero de bandeja
 INPICKER_Handler.DataToSend.ContainerID=10
 INPICKER_Handler.DataToSend.partid=10
 INPICKER_Handler.DataToSend.GraspConfirmation=0
 WAIT SEC 0.2

; DISPARO FOTO
 INPICKER_Handler.DataToSend.command=1

; ESPERA FOTO REALIZADA
 WAIT FOR (INPICKER_Handler.DataReceived.state==15) OR (INPICKER_Handler.DataReceived.state==-1)

IF (INPICKER_Handler.DataReceived.state==-1) THEN

IF (Fallo_nr>=1) THEN
O_INPICKER_OK=FALSE
O_INPICKER_NOK=TRUE

O_TYPE_RQ = FALSE
WAIT FOR I_TYPE_INFO == 0

O_TYPE_RQ = TRUE
WAIT FOR (I_TYPE_INFO >= 1) AND (I_TYPE_INFO <= 5)

SWITCH I_TYPE_INFO

CASE 2
; #### SELECCION DESDE HMI REINTENTO FOTO ####

SELECT_NEXT=FALSE
O_INPICKER_OK=FALSE
O_INPICKER_NOK=FALSE
O_TYPE_RQ = FALSE
GOTO Ini5

CASE 3
; #### SELECCION DESDE HMI CONT SIN CORRECCION ####

SELECT_SIN=TRUE
O_INPICKER_OK=FALSE
O_INPICKER_NOK=TRUE
O_TYPE_RQ = FALSE
GOTO FIN_FOTO5

CASE 4
; #### SELECCION DESDE HMI CERRAR BANDEJA ####
; #### E IR A SIGUIENTE NIVEL             ####

SELECT_NEXT=TRUE
O_INPICKER_OK=FALSE
O_INPICKER_NOK=FALSE
O_TYPE_RQ = FALSE
GOTO FIN_FOTO5

DEFAULT
ENDSWITCH

ELSE

Fallo_nr=Fallo_nr+1
GOTO Ini5

ENDIF
ENDIF

Fin5:
 WAIT SEC 0.1
;ENDFOLD

;FOLD LIN P_FOTO2V_Bandeja5 Vel=0.5 m/s M Tool[5]:T_Camara Base[0];%{PE}%R 8.3.48,%MKUKATPBASIS,%CMOVE,%VLIN,%P 1:LIN, 2:P_FOTO2V_Bandeja5, 3:, 5:0.5, 7:M
$BWDSTART=FALSE
LDAT_ACT=LM
FDAT_ACT=FP_FOTO2V_Bandeja5
BAS(#CP_PARAMS,0.5)
LIN XP_FOTO2V_Bandeja5
;ENDFOLD
;FOLD REALIZA FOTO 2 BANDEJA 5
WAIT SEC 1.0
INPICKER_Handler.DataToSend.GraspConfirmation=1

WAIT FOR (INPICKER_Handler.DataReceived.state==30) OR (INPICKER_Handler.dataReceived.state==-1)

WAIT SEC 0.5

INPICKER_Handler.DataToSend.command=0

IF (INPICKER_handler.datareceived.state==30 ) THEN

IF (INPICKER_Handler.DataReceived.ObjectsGraspable>0) THEN

O_INPICKER_OK=TRUE
O_INPICKER_NOK=FALSE

ELSE

O_INPICKER_OK=FALSE
O_INPICKER_NOK=TRUE

ENDIF

ENDIF

IF (INPICKER_handler.datareceived.state==-1 ) OR (INPICKER_Handler.DataReceived.ObjectsGraspable<=0) THEN

O_INPICKER_OK=FALSE
O_INPICKER_NOK=TRUE

O_TYPE_RQ = FALSE
WAIT FOR I_TYPE_INFO == 0

O_TYPE_RQ = TRUE
WAIT FOR (I_TYPE_INFO >= 1) AND (I_TYPE_INFO <= 5)

SWITCH I_TYPE_INFO

CASE 2
; #### SELECCION DESDE HMI REINTENTO FOTO ####

SELECT_NEXT=FALSE
O_INPICKER_OK=FALSE
O_INPICKER_NOK=FALSE
O_TYPE_RQ = FALSE

IF (INPICKER_Handler.DataReceived.ObjectsGraspable>0)THEN
ELSE
GOTO INICIO_FOTO5
ENDIF

WAIT FOR (INPICKER_Handler.DataReceived.state==0)
GOTO INICIO_FOTO5

CASE 3
; #### SELECCION DESDE HMI CONT SIN CORRECCION ####

SELECT_NEXT=FALSE
O_TYPE_RQ = FALSE

CASE 4
; #### SELECCION DESDE HMI CERRAR BANDEJA ####
; #### E IR A SIGUIENTE NIVEL             ####

SELECT_NEXT=TRUE
O_INPICKER_OK=FALSE
O_INPICKER_NOK=FALSE
O_TYPE_RQ = FALSE

DEFAULT
ENDSWITCH

ENDIF

;ENDFOLD
;FOLD ACTUALIZA BASE DE DESCARGA
FRAMEAUX={X 0,Y 0,Z 0,A 0,B 0,C 0}
FRAME_POS={X 0,Y 0,Z 0,A 0,B 0,C 0}

FRAMEAUX=INPICKER_Handler.DataReceived.PartsToGrasp0.Position
FRAME_POS.x=(FRAMEAUX.x/10)
FRAME_POS.y=(FRAMEAUX.y/10)
FRAME_POS.z=(FRAMEAUX.z/10)
FRAME_POS.a=(FRAMEAUX.a/10)
FRAME_POS.b=(FRAMEAUX.b/10)
FRAME_POS.c=(FRAMEAUX.c/10)

IF FRAME_POS.A < 180.0 THEN
FRAME_POS.A = FRAME_POS.A + 360
ENDIF
IF FRAME_POS.B < 180.0 THEN
FRAME_POS.B = FRAME_POS.B + 360
ENDIF
IF FRAME_POS.A > 180.0 THEN
FRAME_POS.A = FRAME_POS.A - 360
ENDIF
IF FRAME_POS.B > 180.0 THEN
FRAME_POS.B = FRAME_POS.B - 360
ENDIF
FRAME_POS.C = FRAME_POS.C - 360
;ENDFOLD
;FOLD CONTROL LIMITES DE VISION
CTRL_limites()
;ENDFOLD
;FOLD DECISION RESULTADOS EVALUACION BANDEJA 5

IF (O_INPICKER_OK==FALSE) AND (O_INPICKER_NOK==TRUE) THEN
SELECT_NEXT=FALSE
O_TYPE_RQ = FALSE
GOTO FIN_FOTO5
ENDIF


IF (O_LIMITS_OK==FALSE) AND (O_LIMITS_NOK==TRUE) THEN

O_TYPE_RQ = FALSE
WAIT FOR I_TYPE_INFO == 0

O_TYPE_RQ = TRUE
WAIT FOR (I_TYPE_INFO >= 1) AND (I_TYPE_INFO <= 5)

SWITCH I_TYPE_INFO

CASE 2
; #### SELECCION DESDE HMI REINTENTO FOTO ####

SELECT_NEXT=FALSE
O_TYPE_RQ = FALSE
O_LIMITS_OK = FALSE
O_LIMITS_NOK = FALSE
O_LIMIT_X = FALSE
O_LIMIT_Y = FALSE
O_LIMIT_Z = FALSE
O_LIMIT_A = FALSE
O_LIMIT_B = FALSE
O_LIMIT_C = FALSE

GOTO INICIO_FOTO5

CASE 3
; #### SELECCION DESDE HMI CONT SIN CORRECCION ####

SELECT_NEXT=FALSE
O_TYPE_RQ = FALSE

CASE 4
; #### SELECCION DESDE HMI CERRAR BANDEJA ####
; #### E IR A SIGUIENTE NIVEL             ####

SELECT_NEXT=TRUE
O_TYPE_RQ = FALSE
O_LIMITS_OK = FALSE
O_LIMITS_NOK = FALSE
O_LIMIT_X = FALSE
O_LIMIT_Y = FALSE
O_LIMIT_Z = FALSE
O_LIMIT_A = FALSE
O_LIMIT_B = FALSE
O_LIMIT_C = FALSE

DEFAULT

HALT
HALT
HALT
ENDSWITCH

ENDIF
;ENDFOLD
FIN_FOTO5:

DEFAULT
HALT
HALT
; #### SELECCION NO VALIDA ####
HALT
BRAKE

ENDSWITCH

FIN:

;FOLD PTP P20 CONT Vel=50 % M Tool[5]:T_Camara Base[0];%{PE}%R 8.3.48,%MKUKATPBASIS,%CMOVE,%VPTP,%P 1:PTP, 2:P20, 3:C_DIS, 5:50, 7:M
$BWDSTART=FALSE
PDAT_ACT=PM
FDAT_ACT=FP20
BAS(#PTP_PARAMS,50)
PTP XP20 C_DIS
;ENDFOLD

IF (SELECT_NEXT == TRUE) THEN

Rack_Azul_Cerrar_D()

ELSE

;FOLD PTP P30 Vel=50 % M Tool[5]:T_Camara Base[0];%{PE}%R 8.3.48,%MKUKATPBASIS,%CMOVE,%VPTP,%P 1:PTP, 2:P30, 3:, 5:50, 7:M
$BWDSTART=FALSE
PDAT_ACT=PM
FDAT_ACT=FP30
BAS(#PTP_PARAMS,50)
PTP XP30
;ENDFOLD

; POSICION DE SALIDA RACK 2
O_AREL_2=TRUE
ENDIF

;FOLD PTP P40 CONT Vel=50 % PDAT4 Tool[9]:T_Gripper1_Vacio Base[0];%{PE}%R 8.3.48,%MKUKATPBASIS,%CMOVE,%VPTP,%P 1:PTP, 2:P40, 3:C_DIS, 5:50, 7:PDAT4
$BWDSTART=FALSE
PDAT_ACT=PPDAT4
FDAT_ACT=FP40
BAS(#PTP_PARAMS,50)
PTP XP40 C_DIS
;ENDFOLD
END
DEF CTRL_Limites ()

;################################################
; RUTINA DE CONTROL DE LIMITES DE VISION
;
;################################################

IF $T1 THEN
O_LIMITS_OK=FALSE
O_LIMITS_NOK=FALSE
O_LIMIT_X=FALSE
O_LIMIT_Y=FALSE
O_LIMIT_Z=FALSE
O_LIMIT_A=FALSE
O_LIMIT_B=FALSE
O_LIMIT_C=FALSE

LIM_X=FALSE
LIM_Y=FALSE
LIM_Z=FALSE
LIM_A=FALSE
LIM_B=FALSE
LIM_C=FALSE

ELSE

WAIT FOR $EXT
O_LIMITS_OK=FALSE
O_LIMITS_NOK=FALSE
O_LIMIT_X=FALSE
O_LIMIT_Y=FALSE
O_LIMIT_Z=FALSE
O_LIMIT_A=FALSE
O_LIMIT_B=FALSE
O_LIMIT_C=FALSE

LIM_X=FALSE
LIM_Y=FALSE
LIM_Z=FALSE
LIM_A=FALSE
LIM_B=FALSE
LIM_C=FALSE

IF (FRAME_POS.X>-1000.0) AND (FRAME_POS.X<-970.0) THEN
O_LIMIT_X=TRUE
LIM_X=TRUE
ELSE
O_LIMIT_X=FALSE
LIM_X=FALSE
ENDIF

IF (FRAME_POS.Y>1680.0) AND (FRAME_POS.Y<1750.0) THEN
O_LIMIT_Y=TRUE
LIM_Y=TRUE
ELSE
O_LIMIT_Y=FALSE
LIM_Y=FALSE
ENDIF

SWITCH RA_Bandeja_Nr
CASE 21
IF (FRAME_POS.Z>150.0) AND (FRAME_POS.Z<180.0) THEN
O_LIMIT_Z=TRUE
LIM_Z=TRUE
ELSE
O_LIMIT_Z=FALSE
LIM_Z=FALSE
ENDIF
CASE 22
IF (FRAME_POS.Z>360.0) AND (FRAME_POS.Z<385.0) THEN
O_LIMIT_Z=TRUE
LIM_Z=TRUE
ELSE
O_LIMIT_Z=FALSE
LIM_Z=FALSE
ENDIF
CASE 23
IF (FRAME_POS.Z>570.0) AND (FRAME_POS.Z<590.0) THEN
O_LIMIT_Z=TRUE
LIM_Z=TRUE
ELSE
O_LIMIT_Z=FALSE
LIM_Z=FALSE
ENDIF
CASE 24
IF (FRAME_POS.Z>775.0) AND (FRAME_POS.Z<795.0) THEN
O_LIMIT_Z=TRUE
LIM_Z=TRUE
ELSE
O_LIMIT_Z=FALSE
LIM_Z=FALSE
ENDIF
CASE 25
IF (FRAME_POS.Z>975.0) AND (FRAME_POS.Z<1010.0) THEN
O_LIMIT_Z=TRUE
LIM_Z=TRUE
ELSE
O_LIMIT_Z=FALSE
LIM_Z=FALSE
ENDIF
DEFAULT
ENDSWITCH

IF (FRAME_POS.A>88.5) AND (FRAME_POS.A<91.0) THEN
O_LIMIT_A=TRUE
LIM_A=TRUE
ELSE
O_LIMIT_A=FALSE
LIM_A=FALSE
ENDIF

IF (FRAME_POS.B>-2.35) AND (FRAME_POS.B<0.0) THEN
O_LIMIT_B=TRUE
LIM_B=TRUE
ELSE
O_LIMIT_B=FALSE
LIM_B=FALSE
ENDIF

IF (FRAME_POS.C>-180.0) AND (FRAME_POS.C<-179.0) THEN
O_LIMIT_C=TRUE
LIM_C=TRUE
ELSE
O_LIMIT_C=FALSE
LIM_A=FALSE
ENDIF

IF (LIM_X==TRUE) AND (LIM_Y==TRUE) AND (LIM_Z==TRUE) AND (LIM_A==TRUE) AND (LIM_B==TRUE) AND (LIM_C==TRUE) THEN
O_LIMITS_OK=TRUE
O_LIMITS_NOK=FALSE
ELSE
O_LIMITS_OK=FALSE
O_LIMITS_NOK=TRUE
ENDIF
;################################################
ENDIF
END

--- Rack_Azul_Inpicker.dat ---
&ACCESS RVO1
&REL 136
&COMMENT FOTOS EN RACK AZUL
&PARAM EDITMASK = *
&PARAM TEMPLATE = C:\KRC\Roboter\Template\vorgabe
&PARAM DISKPATH = KRC:\R1\Program\MAFELEC
DEFDAT  Rack_Azul_Inpicker
;FOLD EXTERNAL DECLARATIONS;%{PE}%MKUKATPBASIS,%CEXT,%VCOMMON,%P
;FOLD GRIPPERTECH EXT
EXT  H50 (INT  :IN,INT  :IN,INT  :IN,GRP_TYP  :IN )
;ENDFOLD (GRIPPERTECH EXT)
;FOLD SPOTTECH EXT
EXT  USERSPOT (S_COMMAND  :IN,SPOT_TYPE  :IN )
;ENDFOLD (SPOTTECH EXT)
;FOLD BASISTECH EXT;%{PE}%MKUKATPBASIS,%CEXT,%VEXT,%P
EXT  BAS (BAS_COMMAND  :IN,REAL  :IN )
DECL INT SUCCESS
;ENDFOLD (BASISTECH EXT)
;FOLD USER EXT;%{E}%MKUKATPUSER,%CEXT,%VEXT,%P
;Make your modifications here

;ENDFOLD (USER EXT)
;ENDFOLD (EXTERNAL DECLARATIONS)
DECL BASIS_SUGG_T LAST_BASIS={POINT1[] "P0                      ",POINT2[] "P0                      ",CP_PARAMS[] "CPDAT0                  ",PTP_PARAMS[] "PDAT0                   ",CONT[] "                        ",CP_VEL[] "2.0                     ",PTP_VEL[] " 100                    ",SYNC_PARAMS[] "SYNCDAT                 ",SPL_NAME[] "S0                      ",A_PARAMS[] "ADAT0                   "}
DECL PDAT PH={VEL 100.000,ACC 100.000,APO_DIST 100.000,APO_MODE #CDIS,GEAR_JERK 50.0000,EXAX_IGN 0}
DECL PDAT PM={VEL 100.000,ACC 100.000,APO_DIST 100.000,APO_MODE #CDIS,GEAR_JERK 50.0000,EXAX_IGN 0}
DECL E6POS XP_FOTO1V_Bandeja1={X -1356.76111,Y 896.771729,Z 838.201660,A 90.4724884,B 39.6473770,C -91.7588425,S 6,T 19,E1 0.0,E2 0.0,E3 0.0,E4 0.0,E5 0.0,E6 0.0}
DECL FDAT FP_FOTO1V_Bandeja1={TOOL_NO 5,BASE_NO 0,IPO_FRAME #BASE,POINT2[] " ",TQ_STATE FALSE}
DECL E6POS XP_FOTO2V_BANDEJA1={X -727.361816,Y 862.358398,Z 821.780090,A 47.0928421,B 34.4814606,C -110.015610,S 6,T 19,E1 0.0,E2 0.0,E3 0.0,E4 0.0,E5 0.0,E6 0.0}
DECL FDAT FP_FOTO2V_BANDEJA1={TOOL_NO 5,BASE_NO 0,IPO_FRAME #BASE,POINT2[] " ",TQ_STATE FALSE}
DECL E6POS XPOS_ESPERA_FOTO={X -579.686096,Y 282.811523,Z 2283.47388,A 69.3566132,B 20.3452797,C -62.1413918,S 2,T 3,E1 0.0,E2 0.0,E3 0.0,E4 0.0,E5 0.0,E6 0.0}
DECL FDAT FPOS_ESPERA_FOTO={TOOL_NO 5,BASE_NO 0,IPO_FRAME #BASE,POINT2[] " ",TQ_STATE FALSE}
DECL E6POS XP_FOTO1V_Bandeja2={X -1356.75513,Y 896.772888,Z 1000.04065,A 90.4720612,B 39.6473351,C -91.7590103,S 6,T 19,E1 0.0,E2 0.0,E3 0.0,E4 0.0,E5 0.0,E6 0.0}
DECL FDAT FP_FOTO1V_Bandeja2={TOOL_NO 5,BASE_NO 0,IPO_FRAME #BASE,POINT2[] " ",TQ_STATE FALSE}
DECL E6POS XP_FOTO1V_Bandeja3={X -1356.75513,Y 896.772888,Z 1209.91699,A 90.4720612,B 39.6473351,C -91.7590103,S 6,T 19,E1 0.0,E2 0.0,E3 0.0,E4 0.0,E5 0.0,E6 0.0}
DECL FDAT FP_FOTO1V_Bandeja3={TOOL_NO 5,BASE_NO 0,IPO_FRAME #BASE,POINT2[] " ",TQ_STATE FALSE}
DECL E6POS XP_FOTO1V_Bandeja4={X -1356.75513,Y 896.772888,Z 1419.41907,A 90.4720612,B 39.6473351,C -91.7590103,S 6,T 51,E1 0.0,E2 0.0,E3 0.0,E4 0.0,E5 0.0,E6 0.0}
DECL FDAT FP_FOTO1V_Bandeja4={TOOL_NO 5,BASE_NO 0,IPO_FRAME #BASE,POINT2[] " ",TQ_STATE FALSE}
DECL E6POS XP_FOTO1V_Bandeja5={X -1356.75439,Y 896.772461,Z 1667.63367,A 90.4720078,B 39.6473236,C -91.7590,S 6,T 51,E1 0.0,E2 0.0,E3 0.0,E4 0.0,E5 0.0,E6 0.0}
DECL FDAT FP_FOTO1V_Bandeja5={TOOL_NO 5,BASE_NO 0,IPO_FRAME #BASE,POINT2[] " ",TQ_STATE FALSE}
DECL E6POS XP_FOTO2V_Bandeja2={X -727.355530,Y 862.356140,Z 987.705566,A 47.0921135,B 34.4810257,C -110.015305,S 6,T 19,E1 0.0,E2 0.0,E3 0.0,E4 0.0,E5 0.0,E6 0.0}
DECL FDAT FP_FOTO2V_Bandeja2={TOOL_NO 5,BASE_NO 0,IPO_FRAME #BASE,POINT2[] " ",TQ_STATE FALSE}
DECL E6POS XP_FOTO2V_Bandeja3={X -727.348267,Y 862.352722,Z 1189.90515,A 47.0910416,B 34.4808,C -110.015427,S 6,T 51,E1 0.0,E2 0.0,E3 0.0,E4 0.0,E5 0.0,E6 0.0}
DECL FDAT FP_FOTO2V_Bandeja3={TOOL_NO 5,BASE_NO 0,IPO_FRAME #BASE,POINT2[] " ",TQ_STATE FALSE}
DECL E6POS XP_FOTO2V_Bandeja4={X -727.350891,Y 862.353210,Z 1372.38379,A 47.0912323,B 34.4810333,C -110.015900,S 6,T 51,E1 0.0,E2 0.0,E3 0.0,E4 0.0,E5 0.0,E6 0.0}
DECL FDAT FP_FOTO2V_Bandeja4={TOOL_NO 5,BASE_NO 0,IPO_FRAME #BASE,POINT2[] " ",TQ_STATE FALSE}
DECL E6POS XP_FOTO2V_Bandeja5={X -727.355957,Y 862.355652,Z 1582.78748,A 47.0920219,B 34.4812317,C -110.015694,S 6,T 51,E1 0.0,E2 0.0,E3 0.0,E4 0.0,E5 0.0,E6 0.0}
DECL FDAT FP_FOTO2V_Bandeja5={TOOL_NO 5,BASE_NO 0,IPO_FRAME #BASE,POINT2[] " ",TQ_STATE FALSE}
DECL LDAT LM={VEL 2.00000,ACC 20.0000,APO_DIST 100.000,APO_FAC 50.0000,AXIS_VEL 100.000,AXIS_ACC 100.000,ORI_TYP #VAR,CIRC_TYP #BASE,JERK_FAC 50.0000,GEAR_JERK 50.0000,EXAX_IGN 0}
DECL E6POS XP10={X -1012.03430,Y 350.484833,Z 1265.59814,A 97.8802338,B 11.5455894,C -82.2627563,S 6,T 19,E1 0.0,E2 0.0,E3 0.0,E4 0.0,E5 0.0,E6 0.0}
DECL FDAT FP10={TOOL_NO 5,BASE_NO 0,IPO_FRAME #BASE,POINT2[] " ",TQ_STATE FALSE}
DECL E6POS XP20={X -1012.03430,Y 350.484833,Z 1265.59814,A 97.8802338,B 11.5455894,C -82.2627563,S 6,T 19,E1 0.0,E2 0.0,E3 0.0,E4 0.0,E5 0.0,E6 0.0}
DECL FDAT FP20={TOOL_NO 5,BASE_NO 0,IPO_FRAME #BASE,POINT2[] " ",TQ_STATE FALSE}
DECL E6POS XP30={X -579.686096,Y 282.811523,Z 2283.47388,A 69.3566132,B 20.3452797,C -62.1413918,S 2,T 3,E1 0.0,E2 0.0,E3 0.0,E4 0.0,E5 0.0,E6 0.0}
DECL FDAT FP30={TOOL_NO 5,BASE_NO 0,IPO_FRAME #BASE,POINT2[] " ",TQ_STATE FALSE}
DECL E6POS XP1={X -1182.84875,Y -262.316071,Z 1799.99951,A -95.9618378,B 35.3506813,C 86.8218536,S 6,T 26,E1 0.0,E2 0.0,E3 0.0,E4 0.0,E5 0.0,E6 0.0}
DECL FDAT FP1={TOOL_NO 5,BASE_NO 0,IPO_FRAME #BASE,POINT2[] " ",TQ_STATE FALSE}
DECL E6POS XP_ESPERA_FOTO={X -1182.84875,Y -262.316071,Z 1799.99951,A -95.9618378,B 35.3506813,C 86.8218536,S 6,T 26,E1 0.0,E2 0.0,E3 0.0,E4 0.0,E5 0.0,E6 0.0}
DECL FDAT FP_ESPERA_FOTO={TOOL_NO 5,BASE_NO 0,IPO_FRAME #BASE,POINT2[] " ",TQ_STATE FALSE}
DECL PDAT PPDAT1={VEL 100.000,ACC 100.000,APO_DIST 100.000,GEAR_JERK 50.0000,EXAX_IGN 0}
DECL E6POS XP_AFOTO2_B2={X -992.069,Y 757.557495,Z 1057.12793,A 64.1897888,B 38.5717,C -103.388710,S 6,T 19,E1 0.0,E2 0.0,E3 0.0,E4 0.0,E5 0.0,E6 0.0}
DECL FDAT FP_aFOTO2_B2={TOOL_NO 5,BASE_NO 0,IPO_FRAME #BASE,POINT2[] " ",TQ_STATE FALSE}
DECL PDAT PPDAT2={VEL 100.000,ACC 100.000,APO_DIST 100.000,GEAR_JERK 50.0000,EXAX_IGN 0}
DECL E6POS XP_AFOTO1_B2={X -1262.08826,Y 710.299255,Z 1087.34753,A 90.4720612,B 39.6473351,C -91.7590,S 6,T 19,E1 0.0,E2 0.0,E3 0.0,E4 0.0,E5 0.0,E6 0.0}
DECL FDAT FP_aFOTO1_B2={TOOL_NO 5,BASE_NO 0,IPO_FRAME #BASE,POINT2[] " ",TQ_STATE FALSE}
DECL PDAT PPDAT3={VEL 100.000,ACC 100.000,APO_DIST 100.000,GEAR_JERK 50.0000,EXAX_IGN 0}
DECL E6POS XP_AFOTO2_B1={X -1016.78125,Y 770.097839,Z 851.767151,A 66.9011383,B 37.3166046,C -101.599503,S 6,T 19,E1 0.0,E2 0.0,E3 0.0,E4 0.0,E5 0.0,E6 0.0}
DECL FDAT FP_aFOTO2_B1={TOOL_NO 5,BASE_NO 0,IPO_FRAME #BASE,POINT2[] " ",TQ_STATE FALSE}
DECL E6POS XP_AFOTO1_B1={X -1141.63916,Y 731.794189,Z 888.870911,A 90.4710922,B 39.6498184,C -91.7591095,S 6,T 19,E1 0.0,E2 0.0,E3 0.0,E4 0.0,E5 0.0,E6 0.0}
DECL FDAT FP_aFOTO1_B1={TOOL_NO 5,BASE_NO 0,IPO_FRAME #BASE,POINT2[] " ",TQ_STATE FALSE}
DECL E6POS XP_AFOTO1_B3={X -1147.42651,Y 638.023132,Z 1329.99011,A 90.4720612,B 39.6473389,C -91.7590179,S 6,T 51,E1 0.0,E2 0.0,E3 0.0,E4 0.0,E5 0.0,E6 0.0}
DECL FDAT FP_aFOTO1_B3={TOOL_NO 5,BASE_NO 0,IPO_FRAME #BASE,POINT2[] " ",TQ_STATE FALSE}
DECL E6POS XP_AFOTO2_B3={X -1226.82117,Y 745.330750,Z 1244.05371,A 81.1630,B 39.9513626,C -95.9228363,S 6,T 19,E1 0.0,E2 0.0,E3 0.0,E4 0.0,E5 0.0,E6 0.0}
DECL FDAT FP_aFOTO2_B3={TOOL_NO 5,BASE_NO 0,IPO_FRAME #BASE,POINT2[] " ",TQ_STATE FALSE}
DECL E6POS XP_AFOTO1_B4={X -1176.16699,Y 718.736816,Z 1419.19348,A 91.2977066,B 38.0146561,C -91.0080719,S 6,T 51,E1 0.0,E2 0.0,E3 0.0,E4 0.0,E5 0.0,E6 0.0}
DECL FDAT FP_aFOTO1_B4={TOOL_NO 5,BASE_NO 0,IPO_FRAME #BASE,POINT2[] " ",TQ_STATE FALSE}
DECL E6POS XP_AFOTO2_B4={X -924.492859,Y 681.409790,Z 1392.04895,A 65.6965866,B 37.4081039,C -105.465088,S 6,T 51,E1 0.0,E2 0.0,E3 0.0,E4 0.0,E5 0.0,E6 0.0}
DECL FDAT FP_aFOTO2_B4={TOOL_NO 5,BASE_NO 0,IPO_FRAME #BASE,POINT2[] " ",TQ_STATE FALSE}
DECL E6POS XP40={X 288.358063,Y 77.6025696,Z 2718.00244,A -43.7336922,B 54.0647202,C -54.3690681,S 3,T 3,E1 0.0,E2 0.0,E3 0.0,E4 0.0,E5 0.0,E6 0.0}
DECL FDAT FP40={TOOL_NO 9,BASE_NO 0,IPO_FRAME #BASE,POINT2[] " ",TQ_STATE FALSE}
DECL PDAT PPDAT4={VEL 100.000,ACC 100.000,APO_DIST 100.000,APO_MODE #CDIS,GEAR_JERK 50.0000,EXAX_IGN 0}
ENDDAT
